(* CODESYS project DependencyInjectionExport.export

Project tree, tasks and I/O mapping:
  Motors/
    data type e_MotorState
    interface IMotor: Run, Stop, IsRunning
    function block Mock_Motor [ST]: Run, Stop, IsRunning
    function block Motor [ST]: Run, Stop, IsRunning
  function block Machine [ST]
  program PLC_PRG [ST]
*)

// Motors/e_MotorState
TYPE e_MotorState :
(
	Running,
	Stopped,
	Faulted
);
END_TYPE

// Machine
FUNCTION_BLOCK Machine
VAR_INPUT
	Motor : IMotor;
END_VAR
VAR
	RunCondition : BOOL;
END_VAR


IF RunCondition THEN
	Motor.Run();
ELSE
	Motor.Stop();
END_IF

END_FUNCTION_BLOCK

// Motors/Motor
FUNCTION_BLOCK PUBLIC Motor IMPLEMENTS IMotor
VAR_OUTPUT
	Start_Motor : BOOL;
END_VAR
VAR
	State : e_MotorState;
END_VAR

METHOD Run
VAR_INPUT
END_VAR

Start_Motor := TRUE;

State := e_MotorState.Running;
END_METHOD

METHOD Stop
VAR_INPUT
END_VAR

Start_Motor := FALSE;

State := e_MotorState.Stopped;
END_METHOD

PROPERTY IsRunning : BOOL
GET
IsRunning := State = e_MotorState.Running;
END_GET
END_PROPERTY

END_FUNCTION_BLOCK

// Motors/IMotor
INTERFACE IMotor

METHOD Run
VAR_INPUT
END_VAR
END_METHOD

METHOD Stop
VAR_INPUT
END_VAR
END_METHOD

PROPERTY IsRunning : BOOL
GET
END_GET
END_PROPERTY

END_INTERFACE

// PLC_PRG
PROGRAM PLC_PRG
VAR
	MachineA : Machine;
	Mock_MotorA : Mock_Motor;
	MotorA : Motor;
END_VAR


MachineA(Motor := Mock_MotorA);

END_PROGRAM

// Motors/Mock_Motor
FUNCTION_BLOCK PUBLIC Mock_Motor IMPLEMENTS IMotor
VAR
	State : e_MotorState;
END_VAR

METHOD Run
VAR_INPUT
END_VAR

State := e_MotorState.Running;
END_METHOD

METHOD Stop
VAR_INPUT
END_VAR

State := e_MotorState.Stopped;
END_METHOD

PROPERTY IsRunning : BOOL
GET
IsRunning := State = e_MotorState.Running;
END_GET
END_PROPERTY

END_FUNCTION_BLOCK
